// Mitsubishi GX Works2 project: 프로젝트2   PLC: Q02/Q02H

PROGRAM MAIN
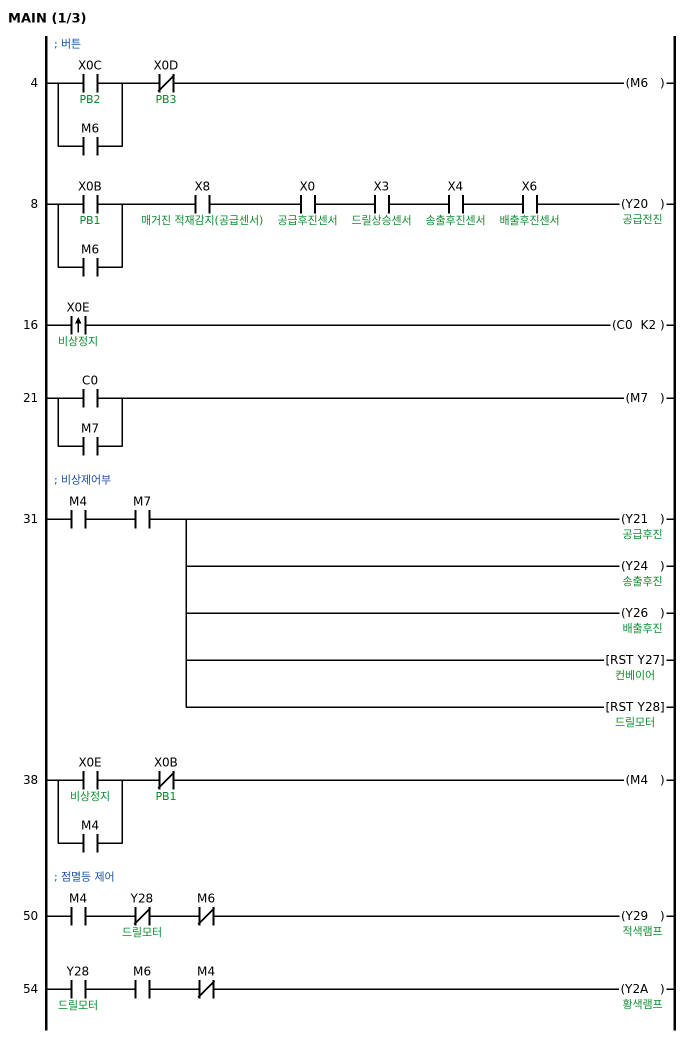
; 버튼
4     LD      X0C  ; PB2
      OR      M6
      ANI     X0D  ; PB3
      OUT     M6
8     LD      X0B  ; PB1
      OR      M6
      AND     X8  ; 매거진 적재감지(공급센서)
      AND     X0  ; 공급후진센서
      AND     X3  ; 드릴상승센서
      AND     X4  ; 송출후진센서
      AND     X6  ; 배출후진센서
      OUT     Y20  ; 공급전진
16    LDP     X0E  ; 비상정지
      OUT     C0 K2
21    LD      C0
      OR      M7
      OUT     M7
; 비상제어부
31    LD      M4
      AND     M7
      OUT     Y21  ; 공급후진
      OUT     Y24  ; 송출후진
      OUT     Y26  ; 배출후진
      RST     Y27  ; 컨베이어
      RST     Y28  ; 드릴모터
38    LD      X0E  ; 비상정지
      OR      M4
      ANI     X0B  ; PB1
      OUT     M4
; 점멸등 제어
50    LD      M4
      ANI     Y28  ; 드릴모터
      ANI     M6
      OUT     Y29  ; 적색램프
54    LD      Y28  ; 드릴모터
      AND     M6
      ANI     M4
      OUT     Y2A  ; 황색램프
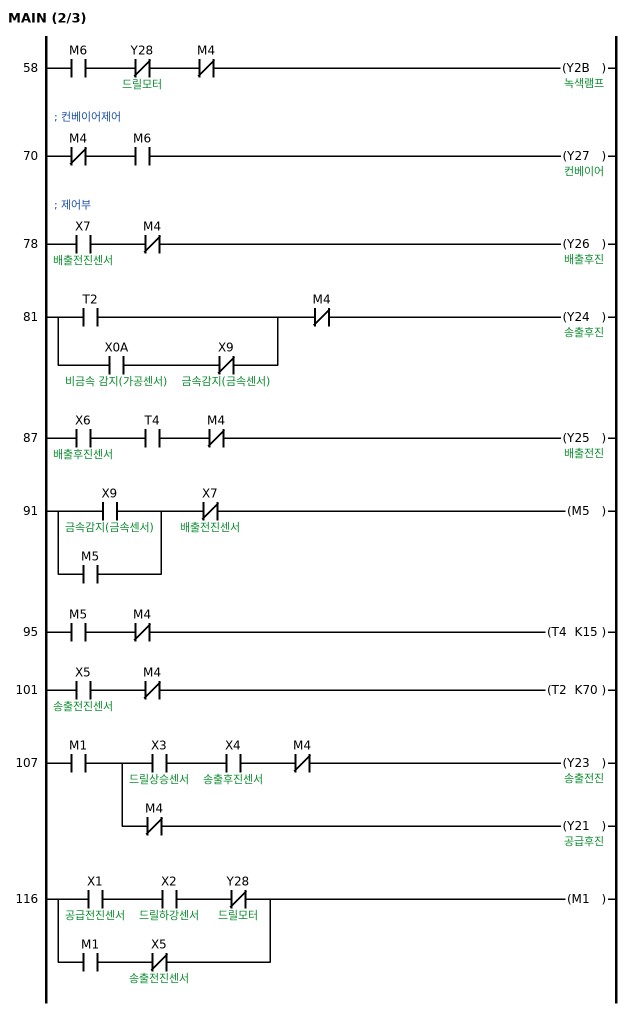
58    LD      M6
      ANI     Y28  ; 드릴모터
      ANI     M4
      OUT     Y2B  ; 녹색램프
; 컨베이어제어
70    LDI     M4
      AND     M6
      OUT     Y27  ; 컨베이어
; 제어부
78    LD      X7  ; 배출전진센서
      ANI     M4
      OUT     Y26  ; 배출후진
81    LD      T2
      LD      X0A  ; 비금속 감지(가공센서)
      ANI     X9  ; 금속감지(금속센서)
      ORB
      ANI     M4
      OUT     Y24  ; 송출후진
87    LD      X6  ; 배출후진센서
      AND     T4
      ANI     M4
      OUT     Y25  ; 배출전진
91    LD      X9  ; 금속감지(금속센서)
      OR      M5
      ANI     X7  ; 배출전진센서
      OUT     M5
95    LD      M5
      ANI     M4
      OUT     T4 K15
101   LD      X5  ; 송출전진센서
      ANI     M4
      OUT     T2 K70
107   LD      M1
      MPS
      AND     X3  ; 드릴상승센서
      AND     X4  ; 송출후진센서
      ANI     M4
      OUT     Y23  ; 송출전진
      MPP
      ANI     M4
      OUT     Y21  ; 공급후진
116   LD      X1  ; 공급전진센서
      AND     X2  ; 드릴하강센서
      ANI     Y28  ; 드릴모터
      LD      M1
      ANI     X5  ; 송출전진센서
      ORB
      OUT     M1
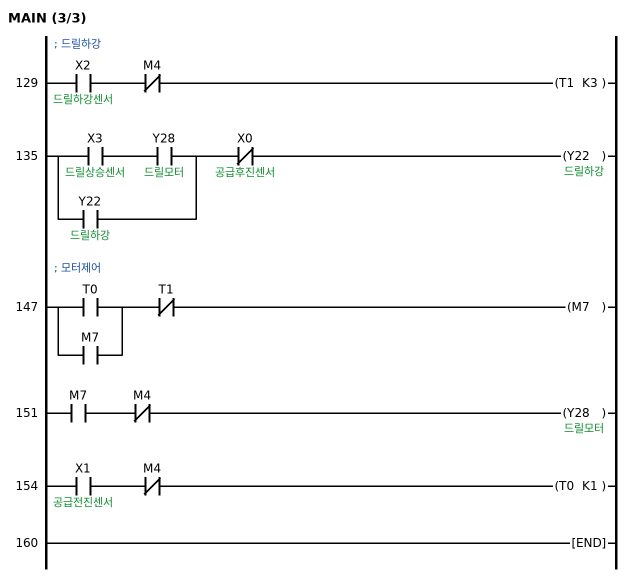
; 드릴하강
129   LD      X2  ; 드릴하강센서
      ANI     M4
      OUT     T1 K3
135   LD      X3  ; 드릴상승센서
      AND     Y28  ; 드릴모터
      OR      Y22  ; 드릴하강
      ANI     X0  ; 공급후진센서
      OUT     Y22  ; 드릴하강
; 모터제어
147   LD      T0
      OR      M7
      ANI     T1
      OUT     M7
151   LD      M7
      ANI     M4
      OUT     Y28  ; 드릴모터
154   LD      X1  ; 공급전진센서
      ANI     M4
      OUT     T0 K1
160   END
END_PROGRAM
